(* LS Electric XG5000 project: ACN_VFD_EIP_FB *)
(* PLC LSPLC *)
(* module base 0 slot 0: Input/Output Module:XEM-DN/DP32HP (DC 24V Input, Transistor Output, 32 Contacts) *)
(* module base 0 slot 1: Internal Positioning:XBF-PO06E (Open Collector Type, 6 Axis) *)
(* module base 0 slot 2: EtherNet/IP:XBL-EIPT (EtherNet/IP communication module, electrical) *)
VAR_GLOBAL
    ACN_VFD_EIP_Input00 : ARRAY[0..3] OF BYTE; (* Input data to ethernet/IP ACN VFD drive *)
    ACN_VFD_EIP_Output00 : ARRAY[0..3] OF BYTE; (* Output data to ethernet/IP ACN VFD drive *)
END_VAR

(* Comments on direct variables
%IX0.0.0	this is comment 1
*)

TYPE ACN_VFD_EIP_UDT : (* this is a user data type for the GS20_Drive_FB *)
STRUCT
    Status_AtReference : BOOL; (* Status of the drive is at the commanded reference *)
    Status_RefFromNet : BOOL; (* Status of that drive is receiving reference from the network. *)
    Status_CtrlFromNet : BOOL; (* Status that control of the drive is from the network. *)
    Status_Ready : BOOL; (* Status that the drive is ready for control. *)
    Status_RunningReverse : BOOL; (* Status that drive is running in reverse direction. *)
    Status_RunningForward : BOOL; (* Status that drive is running in forward direction. *)
    Status_DriveWarning : BOOL; (* Status that there is a drive warning. *)
    Status_DriveFaulted : BOOL; (* Status that drive is faulted. *)
    Status_DriveState : SINT; (* Status of drive state. *)
    Status_CurrentReferenceHz : REAL; (* Current speed reference of the drive in Hz. *)
    Cmd_FaultReset : BOOL; (* Reset drive fault *)
    Cmd_RunReverse : BOOL; (* Command to run in reverse direction. *)
    Cmd_RunForward : BOOL; (* Command to run in forward direction. *)
    Cmd_SpeedReferenceHz : REAL; (* Command speed reference in Hz *)
END_STRUCT;
END_TYPE

FUNCTION_BLOCK ACN_VFD_EIP_FB
(* This function block is used to control and receive status of a ACN inverter drive. *)
VAR_INPUT
    Enable : BOOL; (* Enable the function block. *)
    InputData : ARRAY[0..3] OF BYTE; (* Ethernet/IP input data array *)
END_VAR
VAR_IN_OUT
    ACN_User_UDT : ACN_VFD_EIP_UDT; (* User data type variable for controlling ACN VFD *)
    OutputData : ARRAY[0..3] OF BYTE; (* Ethernet/IP output data array *)
END_VAR
VAR_OUTPUT
    Active : BOOL; (* Status that function block is enabled. *)
END_VAR
VAR
    BTempInput : ARRAY[0..3] OF BYTE; (* temporary byte array *)
    BTempOutput : ARRAY[0..3] OF BYTE; (* temporary byte array *)
    ITemp : INT; (* temporary int value *)
    Temporary_Word : WORD; (* temporary word storage *)
END_VAR
(***************************************************************************************************
(* 
AutomationDirect.com has provided this code for convenience. This sample code is provided "as-is" with no expressed or implied warranty. 
 If the end user includes any of the sample code (in whole or part), it is the user's responsibility to completely modify, integrate, and test any code to ensure it meets all system and 
 safety requirements for the intended application or system.
 

	The 'ACN_VFD_EIP_FB' function block uses data type BYTE for the InputData and OutputData.
		When creating a new module using the EDS file, select the data type BYTE.
		
									Data type:: BYTE
									Input Size: 4 BYTES
									Output Size: 4 BYTES
									EDS File: IronHorse_ACN-ETH_Rev1_2.eds
									
	***************************************************************************************************)
	
IF (Enable = TRUE) THEN		
	Active := TRUE;	
	
	(***********************
  	Mapping Input Data 
  	***********************)
  	
  	BTempInput :=ARY_MOVE(MOVE_NUM:=4, IN:=InputData, IN_INDX:=0, OUT_INDX:=0);	
  	
 	ACN_User_UDT.Status_DriveFaulted := BTempInput[0].0;
	ACN_User_UDT.Status_DriveWarning := BTempInput[0].1;
  	ACN_User_UDT.Status_RunningForward := BTempInput[0].2;
	ACN_User_UDT.Status_RunningReverse:= BTempInput[0].3;
	ACN_User_UDT.Status_Ready := BTempInput[0].4;
	ACN_User_UDT.Status_CtrlFromNet := BTempInput[0].5;
	ACN_User_UDT.Status_RefFromNet := BTempInput[0].6;
	ACN_User_UDT.Status_AtReference := BTempInput[0].7;


	//drive state
	ACN_User_UDT.Status_DriveState := BYTE_TO_SINT(IN:=BTempInput[1]);
	
	//Status for Drive Speed in HZ
	Temporary_Word := BYTE_WORD(LOW:=BTempInput[2], HIGH:=BTempInput[3]);
	ITemp := WORD_TO_INT(IN:=Temporary_Word);
	ACN_User_UDT.Status_CurrentReferenceHz :=  INT_TO_REAL(IN:=ITemp)  / 100.0;
	
	
	(***********************
  	Mapping Output Data 
  	***********************)
 	BTempOutput[0].0 := ACN_User_UDT.Cmd_RunForward;
 	BTempOutput[0].1 := ACN_User_UDT.Cmd_RunReverse;
 	BTempOutput[0].2 := ACN_User_UDT.Cmd_FaultReset;
 	
 	//CMD for Drive Speed in HZ
	ITemp :=  REAL_TO_INT(ACN_User_UDT.Cmd_SpeedReferenceHz * 100.0);
	Temporary_Word := INT_TO_WORD(IN:=ITemp);
 	WORD_BYTE(IN:=Temporary_Word, LOW=>BTempOutput[2], HIGH=>BTempOutput[3]);
 
 	
 	OutputData :=ARY_MOVE(MOVE_NUM:=4, IN:=BTempOutput, IN_INDX:=0, OUT_INDX:=0);


ELSE
	Active := FALSE;
END_IF;
END_FUNCTION_BLOCK

PROGRAM FB_Usage_LD (* task: Scan Program *)
VAR
    ACN_FB_INST_00 : ACN_VFD_EIP_FB;
    ACN_VFD_00 : ACN_VFD_EIP_UDT;
    fbActive : BOOL;
END_VAR
VAR_EXTERNAL
    ACN_VFD_EIP_Input00 : ARRAY[0..3] OF BYTE; (* Input data to ethernet/IP ACN VFD drive *)
    ACN_VFD_EIP_Output00 : ARRAY[0..3] OF BYTE; (* Output data to ethernet/IP ACN VFD drive *)
END_VAR

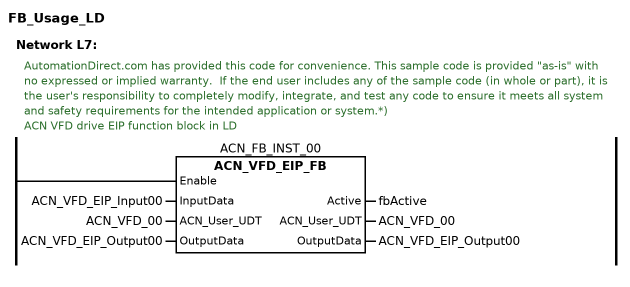
(* AutomationDirect.com has provided this code for convenience. This sample code is provided "as-is" with no expressed or implied warranty.  If the end user includes any of the sample code (in whole or part), it is the user's responsibility to completely modify, integrate, and test any code to ensure it meets all system and safety requirements for the intended application or system.* ) *)
(* ACN VFD drive EIP function block in LD *)
(* Rung L7 *)
ACN_FB_INST_00(Enable := TRUE, InputData := ACN_VFD_EIP_Input00, ACN_User_UDT := ACN_VFD_00, OutputData := ACN_VFD_EIP_Output00, Active => fbActive, ACN_User_UDT => ACN_VFD_00, OutputData => ACN_VFD_EIP_Output00);
END_PROGRAM

PROGRAM FB_Usage_ST (* task: Scan Program *)
(*  *)
VAR
    ACN_INST_00 : ACN_VFD_EIP_FB;
    ACN_VFD_00 : ACN_VFD_EIP_UDT;
    fbActive : BOOL;
    ITemp : INT;
END_VAR
VAR_EXTERNAL
    ACN_VFD_EIP_Input00 : ARRAY[0..3] OF BYTE; (* Input data to ethernet/IP ACN VFD drive *)
    ACN_VFD_EIP_Output00 : ARRAY[0..3] OF BYTE; (* Output data to ethernet/IP ACN VFD drive *)
END_VAR
(* 
AutomationDirect.com has provided this code for convenience. This sample code is provided "as-is" with no expressed or implied warranty. 
 If the end user includes any of the sample code (in whole or part), it is the user's responsibility to completely modify, integrate, and test any code to ensure it meets all system and 
 safety requirements for the intended application or system.
 *)



fbActive := TRUE;

//ACN_INST_00(Enable:=TRUE, InputData:=ACN_VFD_EIP_Input00, ACN_User_UDT:=ACN_VFD_00, OutputData:=ACN_VFD_EIP_Output00, Active=>fbActive);
END_PROGRAM